TYPE St_Assy_GetDetails EXTENDS St_Assy_Base :
STRUCT
END_STRUCT
END_TYPE

(* stored: Version 1.1.0.1, ProductVersion 3.1.4024.12
   DUT St_Assy_GetDetails: Id {92d2ceb5-5196-4599-86aa-a09ece036572} *)
